// TIA Portal V17 export
// export: Created 2024-06-14T09:53:04.9403507Z, ExportSetting WithDefaults, DisplayName Totally Integrated Automation Portal, DisplayVersion V17, DisplayName TIA Portal Openness, DisplayVersion V17, DisplayName TIA Portal Version Control Interface, DisplayVersion V17, DisplayName Simotion SCOUT TIA, DisplayVersion 5.4.3.0, DisplayName SINAMICS Startdrive Advanced, DisplayVersion V17 SP1 Update 1, DisplayName SINAMICS Startdrive G110M, G120, G120C, G120D, G120P, G115D, DisplayVersion V17 SP1 Update 1, DisplayName SINAMICS Startdrive G130, G150, S120, S150, SINAMICS MV, S210, DisplayVersion V17 SP1 Update 1, DisplayName STEP 7 Professional, DisplayVersion V17, DisplayName STEP 7 Safety, DisplayVersion V17, DisplayName WinCC Professional, DisplayVersion V17
DATA_BLOCK "keypad_logic_DB"   // DB4
VERSION : 0.1
// stored: AutoNumber true, DBAccessibleFromOPCUA true, InstanceOfName keypad_logic, InstanceOfType FB
"keypad_logic"
   // VAR_INPUT
   //    Num_0 : Bool;
   //    Num_1 : Bool;
   //    Num_2 : Bool;
   //    Num_3 : Bool;
   //    Num_4 : Bool;
   //    Num_5 : Bool;
   //    Num_6 : Bool;
   //    Num_7 : Bool;
   //    Num_8 : Bool;
   //    Num_9 : Bool;
   //    enter : Bool;
   //    clear : Bool;
   // END_VAR
   // VAR
   //    count_0 : CTU_INT;
   // END_VAR
   // VAR RETAIN
   //    Tens { S7_SetPoint := 'True'} : Int;
   // END_VAR
   // VAR
   //    ones : Int;
   //    decimal : Int;
   //    P_TRIG : Bool;
   //    MUL : Int;
   //    MUL_1 : Int;
   //    Tare_weight : Real;
   //    "count _reset" : Bool;
   //    Tare_Entry : Real;
   //    "screen count" : Int;
   //    screen_number : Int;
   //    screen_reset : Bool;
   //    MUL_2 : Int;
   //    count_1 : CTU_INT;
   //    count_cv_1 : Int;
   //    "BPCL COUNT" : Int;
   //    DOMESTIC : Bool;
   //    COMMERCIAL : Bool;
   //    MALALBAR_COUNT : Int;
   // END_VAR
   // VAR RETAIN
   //    SENSE_1 : Int;
   //    SENSE_2 : Int;
   //    SENSE_3 : Int;
   //    SENSE_4 : Int;
   // END_VAR
   // VAR
   //    "SENSI NG_TIME" : Int;
   //    sens_reset : Bool;
   //    "open screen" : Bool;
   //    DOMESTIC_1 : Bool;
   //    COMMERCIAL_1 : Bool;
   //    count_2 : CTU_INT;
   // END_VAR
   // VAR RETAIN
   //    password { S7_SetPoint := 'True'} : Int;
   // END_VAR
   // VAR
   //    password_1 : Int;
   //    password_2 : Int;
   //    password_3 : Int;
   //    password_4 : Int;
   //    password_5 : Int;
   //    mul_3 : Int;
   //    mul_4 : Int;
   //    mul_5 : Int;
   //    mul_6 : Int;
   //    password_reset : Bool;
   //    sens : Bool;
   // END_VAR
BEGIN
END_DATA_BLOCK
